// TIA Portal V20 export
// export: Created 2025-12-01T14:56:14.2542471Z, ExportSetting None, DisplayName Totally Integrated Automation Portal, DisplayVersion V20 Update 3, DisplayName TIA Portal Openness, DisplayVersion V20 Update 3, DisplayName TIA Portal Version Control Interface, DisplayVersion V20 Update 3, DisplayName STEP 7 Professional, DisplayVersion V20 Update 3, DisplayName STEP 7 Safety, DisplayVersion V20 Update 2, DisplayName WinCC Basic/Comfort/Advanced, DisplayVersion V20 Update 3, DisplayName WinCC Professional, DisplayVersion V20 Update 3, DisplayName WinCC Unified, DisplayVersion V20 Update 3
TYPE "UDT_UTs_DatosQUBIQA"
   STRUCT
      PID : Array[0..19] of Char;   // PID
      NumeroDeBulto : UInt;   // Numero de Bulto
      TotalBultos : UInt;   // Numero Total de Bultos
      LongitudPID : UInt;   // Longitud del PID
   END_STRUCT;
END_TYPE
